FUNCTION_BLOCK FB_MKS_925
VAR_INPUT
	stVolume : ST_Volume;
	q_xGaugeConnected	:	BOOL;
END_VAR
VAR_OUTPUT
END_VAR
VAR_IN_OUT
	stGauge	:	ST_MKS_925;
END_VAR
VAR
END_VAR

(* 
MKS 925 Vacuum gauge

A vacuum gauge takes as input, the pressure of the volume it is attached to,
and produces on its analog output, a corresponding voltage.


*)

IF q_xGaugeConnected THEN
	(*set gauge real pressure based on chamber real pressure*)
	stGauge.rPress := stVolume.rPressure;
	(*set gauge raw pressure based on transformation of real pressure*)
	stGauge.q_iRawPress := F_MKS_925(stGauge);// gauge on
ELSE
	stGauge.rPress := 0;
	stGauge.q_iRawPress := 0; // gauge not on ??
END_IF

END_FUNCTION_BLOCK

(* stored: Version 1.1.0.1, ProductVersion 3.1.4020.12
   POU FB_MKS_925: Id {326e9f8e-ca6d-499b-833c-5f81933531e2}, SpecialFunc None *)
